Staubli VAL3: MotionPage.dtx

mdesc mNomSpeed = {leave=5, reach=5}
num nAxisNum = 6
bool bHomeDone
bool bAlignDone
mdesc mjoint = {blend=cartesian}
